TYPE TFMachinePalletizer_Zone :
STRUCT
	
	WorkArea	: ARRAY[1..MAXAREA] OF INT; 			(* Numero delle WorkArea *)
	Code		: ARRAY[1..MAXFORMINGCODE] OF INT;		(* Codici di Pallettizzazione (0..n=, -1 dato non valido) *)
	
END_STRUCT
END_TYPE

(* stored: Version 1.1.0.1, ProductVersion 3.1.4024.11
   DUT TFMachinePalletizer_Zone: Id {4f6ee5fa-51bb-4671-8efa-90fce237bf7b} *)
